Fanuc KAREL source: ka00089.KL

PROGRAM KA00089
%STACKSIZE=65535
%PRIORITY=65535
%NOLOCKGROUP
VAR
SRC : JOINTPOS9
DST : POSITION
BEGIN
-- UNSAFE_SOURCE_IR line 7: DST = convert_jointpos9_to_position(SRC)
END KA00089
